// TwinCAT 3 PLC project HelloWorldPLC
// ProgramVersion: 3.1.4024.0
// libraries:
//   Tc2_Standard, * (Beckhoff Automation GmbH)
//   Tc2_System, * (Beckhoff Automation GmbH)
//   Tc3_Module, * (Beckhoff Automation GmbH)
// project tree:
//   DUTs/ E_Color.TcDUT
//   / PlcTask.TcTTO
//   POUs/ MAIN.TcPOU

CONFIGURATION HelloWorldPLC
    RESOURCE PLC ON TwinCAT3
        TASK PlcTask(INTERVAL := T#10ms, PRIORITY := 6);
        PROGRAM MAIN WITH PlcTask : MAIN;
    END_RESOURCE
END_CONFIGURATION

// ---- DUTs/E_Color.TcDUT
{attribute 'qualified_only'}
{attribute 'strict'}
TYPE E_Color :
(
	enum_member := 0
);
END_TYPE

// ---- POUs/MAIN.TcPOU
PROGRAM MAIN
VAR
	bRunOnlyOnce : BOOL := FALSE;
END_VAR

IF NOT bRunOnlyOnce THEN
		ADSLOGSTR(msgCtrlMask := ADSLOG_MSGTYPE_ERROR OR ADSLOG_MSGTYPE_LOG, 
			msgFmtStr := 'Hello',
			strArg :='');
		bRunOnlyOnce := TRUE;
END_IF

END_PROGRAM
